// TwinCAT 3 PLC project ECRH
// ProgramVersion: 3.1.4023.0
// libraries:
//   Tc2_MBus, * (Beckhoff Automation GmbH)
//   Tc2_MC2, * (Beckhoff Automation GmbH)
//   Tc2_NC, * (Beckhoff Automation GmbH)
//   Tc2_Standard, * (Beckhoff Automation GmbH)
//   Tc2_System, * (Beckhoff Automation GmbH)
//   Tc3_Module, * (Beckhoff Automation GmbH)
// project tree:
//   GVLs/ GVL.TcGVL
//   / PlcTask.TcTTO
//   POUs/ MAIN.TcPOU, MAP.TcPOU, pCTRL_CODAC.TcPOU

CONFIGURATION ECRH
    RESOURCE PLC ON TwinCAT3
        TASK PlcTask(INTERVAL := T#10ms, PRIORITY := 20);
        PROGRAM MAIN WITH PlcTask : MAIN;
    END_RESOURCE
END_CONFIGURATION

// ---- GVLs/GVL.TcGVL
{attribute 'qualified_only'}
VAR_GLOBAL
	// Constantes de contrôle à ne pas dépasser
	dTemperature_Seuil_TBD : LREAL := 80000;
	dTension_Max : LREAL := 300;
	dCouple_Max : LREAL := 63 (*0.75 * 100 / 1.2*);
	
	// Peut-être à remplacer par les limites d'axes à définir dans MOTION -> Axes -> limit switches
	Butee_Min_M1X : LREAL := -49;
	Butee_Min_M1Y : LREAL := -17;
	Butee_Min_M2X : LREAL := -100;
	Butee_Min_M2Y : LREAL := -100;
	Butee_Min_M3X : LREAL := -100;
	Butee_Min_M3Y : LREAL := -100;
	Butee_Max_M1X : LREAL := 39;
	Butee_Max_M1Y : LREAL := 16;
	Butee_Max_M2X : LREAL := 100;
	Butee_Max_M2Y : LREAL := 100;
	Butee_Max_M3X : LREAL := 100;
	Butee_Max_M3Y : LREAL := 100;
	
	// Variable d'erreurs à envoyer au codac à intervalles de temps réguliers
	arrErrorSystem : ARRAY[0..4] OF BOOL := [FALSE, FALSE, FALSE, FALSE, FALSE];
	arrErrorTemperature : ARRAY[0..5] OF BOOL := [FALSE, FALSE, FALSE, FALSE, FALSE, FALSE];
	arrErrorTension : ARRAY[0..2] OF BOOL := [FALSE, FALSE, FALSE];
	arrErrorCouple : ARRAY[0..5] OF BOOL := [FALSE, FALSE, FALSE, FALSE];
	arrErrorPosition : ARRAY[0..5] OF BOOL := [FALSE, FALSE, FALSE, FALSE];
	
	// Variable qui stocke l'état de la commande moteur
	iEtatCmd : INT := 0;
	
	// Initialise la vitesse des moteurs
	dVelocite : LREAL := 10;
	dAcceleration : LREAL := 2;
	dDeceleration : LREAL := 2;
	dJerk : LREAL := 5000;
	
	// Définition des axes, doit être link aux axes du motion control
	M1_X : AXIS_REF;
	M1_Y : AXIS_REF;
	M2_X : AXIS_REF;
	M2_Y : AXIS_REF;
	M3_X : AXIS_REF;
	M3_Y : AXIS_REF;
	
	// Variable qui indique si une erreur est remarquée sur le système
	bError : BOOL := FALSE;
	
	// Variable qui définit la position voulue par le PCS
	dSetPosition_M1X : LREAL;
	dSetPosition_M1Y : LREAL;
	dSetPosition_M2X : LREAL;
	dSetPosition_M2Y : LREAL;
	dSetPosition_M3X : LREAL;
	dSetPosition_M3Y : LREAL;
	
	// Variable qui retient si une erreur est survenue lors de la dernière commande
	bErrorTwincat : BOOL;
	
	// Variable dont la valeur correspond à celle mesurée par le ThermoCouple indiqué
	arrTemperatures : ARRAY[0..5] OF LREAL;
	iTC1_M1 AT %I* : INT := 0;
	iTC2_M1 AT %I* : INT := 0;
	iTC1_M2 AT %I* : INT := 0;
	iTC2_M2 AT %I* : INT := 0;
	iTC1_M3 AT %I* : INT := 0;
	iTC2_M3 AT %I* : INT := 0;
		
	// Variable dont la valeur correspond à celle mesurée par le capteur de tension du câble
	arrTensions : ARRAY[0..2] OF LREAL;
	iTension_M1 AT %I* : INT := 0;
	iTension_M2 AT %I* : INT := 0;
	iTension_M3 AT %I* : INT := 0;
		
	// Variable à remplacer par la vrai variable qui indique si les moteurs sont arrêtés
	bMotor_Stopped : BOOL := FALSE;
	
	// Buffer qui contient les données d'intérêt des 200 dernières ms, ms étant l'index correspondant à la ms de l'instant t
	arrData : ARRAY [0..199] OF ARRAY[0..14] OF LREAL;
	ms : INT := 0;
	
	// Tableaux de données destinés à êtres récupérés par le CODAC -> faciliter l'accès aux données
	arrValues : ARRAY[0..14] OF LREAL;
	arrErrors : ARRAY[0..14] OF BOOL;
	arrButees : ARRAY[0..11] OF LREAL;
	
	// Détecteur placé proche de la butée mécanique pour permettre le homing de la position et avoir à partir de ce point un mouvement relatif connu
	bHomeSwitch_M1X AT %I*: BOOL;
	bHomeSwitch_M1Y AT %I*: BOOL;
	bHomeSwitch_M2X AT %I*: BOOL;
	bHomeSwitch_M2Y AT %I*: BOOL;
	bHomeSwitch_M3X AT %I*: BOOL;
	bHomeSwitch_M3Y AT %I*: BOOL;
	
	// Définit le mouvement à faire pour retomber sur une consigne moteur correspondant au 0° à partir de la position de homing
	dZero_M1X: LREAL;
	dZero_M1Y: LREAL;
	dZero_M2X: LREAL;
	dZero_M2Y: LREAL;
	dZero_M3X: LREAL;
	dZero_M3Y: LREAL;
	
	// Définit la commande de couple de chaque axe
	dSetTorque_M1X AT %Q*: UINT := 62;
	dSetTorque_M1Y AT %Q*: UINT := 62;
	dSetTorque_M2X AT %Q*: UINT := 62;
	dSetTorque_M2Y AT %Q*: UINT := 62;
	dSetTorque_M3X AT %Q*: UINT := 62;
	dSetTorque_M3Y AT %Q*: UINT := 62;
	
	// Boolean qui indique si l'initialisation est bien réalisée 
	bInit_OK: BOOL;

END_VAR

// ---- POUs/MAIN.TcPOU
PROGRAM MAIN
VAR
	Initialisation: INT := 0;
	En_Attente: INT := 100;
	En_Cours_De_Traitement: INT := 200;
	Stop: INT := 300;
	Reset: INT := 800;
	Erreur: INT := 900;
	
	McPower_M1X : MC_Power;
	McReset_M1X : MC_Reset;
	McStop_M1X : MC_Stop;
	McHome_M1X : MC_Home;
	McMoveAbs_M1X : MC_MoveAbsolute;
	
	McPower_M1Y : MC_Power;
	McReset_M1Y : MC_Reset;
	McStop_M1Y : MC_Stop;
	McHome_M1Y : MC_Home;
	McMoveAbs_M1Y : MC_MoveAbsolute;
END_VAR

// A chaque itération, il faut penser à appeler la fonction pour que son statut (Done, Busy, Error) se mette à jour
// Une façon de faire est d'appeler au début chaque fonction et de changer dans le corps du programme
// seulement le execute qui vaut true ou false
GVL.M1_X.ReadStatus();
McPower_M1X(Axis:=GVL.M1_X,Enable:=TRUE,Enable_Positive:=TRUE,Enable_Negative:=TRUE,Override:=100);
McReset_M1X(Axis:=GVL.M1_X);
McHome_M1X(Axis:=GVL.M1_X,bCalibrationCam := GVL.bHomeSwitch_M1X);
McMoveAbs_M1X(Axis:=GVL.M1_X);
McStop_M1X(Axis:=GVL.M1_X);

GVL.M1_Y.ReadStatus();
McPower_M1Y(Axis:=GVL.M1_Y,Enable:=TRUE,Enable_Positive:=TRUE,Enable_Negative:=TRUE,Override:=100);
McReset_M1Y(Axis:=GVL.M1_Y);
McHome_M1Y(Axis:=GVL.M1_Y,bCalibrationCam := GVL.bHomeSwitch_M1Y);
McMoveAbs_M1Y(Axis:=GVL.M1_Y);
McStop_M1Y(Axis:=GVL.M1_Y);

// Permet d'actualiser les données qui vont transités par ADS vers le CODAC
pCTRL_CODAC();

CASE GVL.iEtatCmd OF

	// INITIALISATION
	0: 
		// On commence par tout disable pour être sûr qu'il n'y ait pas d'erreur
		McReset_M1X(Axis:=GVL.M1_X, Execute:=FALSE);
		McHome_M1X(Axis:=GVL.M1_X,bCalibrationCam := GVL.bHomeSwitch_M1X, Execute:=FALSE);
		McMoveAbs_M1X(Axis:=GVL.M1_X, Execute:=FALSE);
		McStop_M1X(Axis:=GVL.M1_X, Execute:=FALSE);
		
		McReset_M1Y(Axis:=GVL.M1_Y, Execute:=FALSE);
		McHome_M1Y(Axis:=GVL.M1_Y,bCalibrationCam := GVL.bHomeSwitch_M1Y, Execute:=FALSE);
		McMoveAbs_M1Y(Axis:=GVL.M1_Y, Execute:=FALSE);
		McStop_M1Y(Axis:=GVL.M1_Y, Execute:=FALSE);
		
		// L'initialisation n'est pas faite donc on assigne FALSE
		GVL.bInit_OK := FALSE;
	
		// On commence par lancer un reset des axes
		McReset_M1X(Axis:= GVL.M1_X, Execute:= TRUE);
		McReset_M1Y(Axis:= GVL.M1_Y, Execute:= TRUE);
		IF GVL.bError OR McReset_M1X.Error OR McReset_M1Y.Error THEN
			GVL.iEtatCmd := Erreur;
		ELSE
			GVL.iEtatCmd := 5;				
		END_IF
		
		// On assigne au tableau de butées les valeurs à récupérer au CODAC
		GVL.arrButees[0]:=GVL.Butee_Min_M1X;
		GVL.arrButees[1]:=GVL.Butee_Max_M1X;
		GVL.arrButees[2]:=GVL.Butee_Min_M1Y;
		GVL.arrButees[3]:=GVL.Butee_Max_M1Y;
		GVL.arrButees[4]:=GVL.Butee_Min_M2X;
		GVL.arrButees[5]:=GVL.Butee_Max_M2X;
		GVL.arrButees[6]:=GVL.Butee_Min_M2Y;
		GVL.arrButees[7]:=GVL.Butee_Max_M2Y;
		GVL.arrButees[8]:=GVL.Butee_Min_M3X;
		GVL.arrButees[9]:=GVL.Butee_Max_M3X;
		GVL.arrButees[10]:=GVL.Butee_Min_M3Y;
		GVL.arrButees[11]:=GVL.Butee_Max_M3Y;
	
	// On attend la fin du reset
	5: 
		IF GVL.bError OR McReset_M1X.Error OR McReset_M1Y.Error THEN
			GVL.iEtatCmd := Erreur;
		ELSIF McReset_M1X.Done AND McReset_M1Y.Done THEN
			 GVL.iEtatCmd := 20;		
			McReset_M1X(Axis:= GVL.M1_X, Execute:= FALSE);
			McReset_M1Y(Axis:= GVL.M1_Y, Execute:= FALSE);		
		END_IF
		
	(* 10 réservée à la commande de limitation de couple originellement
	   finalement, celle-ci se réalise directement via la variable globale SetTorque
	   qui est linkée à bipolar torque limit au niveau du drive *)

	// On lance un homing général qui met le système au niveau du point connu avec la distance adaptée. 
	// La première fois, faire le homing jusqu'à 0 et déplacer le moteur jusqu'à la position de 0°
	// Configurer cette distance dans la calibration value sous M1_X -> Enc -> Homing -> Calibration value
	// Le 0 absolu est maintenant configuré au niveau du 0° et le homing arrive à -Dist
	20: 
		McHome_M1X(Axis:=GVL.M1_X, Execute:= TRUE, bCalibrationCam := GVL.bHomeSwitch_M1X, Position:= GVL.dZero_M1X);
		McHome_M1Y(Axis:=GVL.M1_Y, Execute:= TRUE, bCalibrationCam := GVL.bHomeSwitch_M1Y, Position:= GVL.dZero_M1Y);
		IF GVL.bError OR McHome_M1X.Error OR McHome_M1Y.Error THEN
			GVL.iEtatCmd := 900;
		ELSE
			GVL.iEtatCmd := 25;
		END_IF
			
	// On attend la fin du homing
	25: 
		IF McHome_M1Y.Error OR McHome_M1X.Error OR GVL.bError THEN
			GVL.iEtatCmd := Erreur;
		ELSIF McHome_M1X.Done AND McHome_M1Y.Done THEN
			McHome_M1X(Axis:= GVL.M1_X, Execute:= FALSE);
			McHome_M1Y(Axis:= GVL.M1_Y, Execute:= FALSE);
			GVL.iEtatCmd := 30;		
		END_IF
		
	// On fait un mouvement vers le 0 absolu  -- Seulement si la calibration value ne marche pas (30 à 50 inutile normalement)
	30: 
		McMoveAbs_M1X(Axis:=GVL.M1_X,
					Position:= 0,
					Velocity:= GVL.dVelocite,
					Acceleration:= GVL.dAcceleration,
					Deceleration:= GVL.dDeceleration,
					Jerk:= GVL.dJerk,
					Execute:= TRUE);
		McMoveAbs_M1Y(Axis:=GVL.M1_Y,
					Position:= 0,
					Velocity:= GVL.dVelocite,
					Acceleration:= GVL.dAcceleration,
					Deceleration:= GVL.dDeceleration,
					Jerk:= GVL.dJerk,
					Execute:= TRUE);
		IF GVL.bError OR McMoveAbs_M1X.Error OR McMoveAbs_M1Y.Error THEN
			GVL.iEtatCmd := 900;
		ELSE
			GVL.iEtatCmd := 35;
		END_IF
	
	35: // On attend le mouvement vers le 0 absolu
		IF McMoveAbs_M1Y.Error OR McMoveAbs_M1X.Error OR GVL.bError THEN
			GVL.iEtatCmd := Erreur;
		ELSIF McMoveAbs_M1X.Done AND McMoveAbs_M1Y.Done THEN
			McMoveAbs_M1X(Axis:= GVL.M1_X, Execute:= FALSE);
			McMoveAbs_M1Y(Axis:= GVL.M1_Y, Execute:= FALSE);
			GVL.bInit_OK:= TRUE;
			GVL.iEtatCmd := En_Attente;		
		END_IF
	
	100: // En attente d'un changement induit en ADS ou d'une erreur
		IF GVL.bError THEN
			GVL.iEtatCmd := Erreur;
		END_IF
		
	// Entâme de la phase de mouvement moteur : 
	// Déplacement moteur miroir en premier hors butees (PAS FORCEMENT NECESSAIRE) 
	// Déplacement cadre vers position voulue
	// Deplacement miroir vers position voulue
	// Retour en phase d'attente
	200:
		McMoveAbs_M1Y(Axis:=GVL.M1_Y,
					Position:= 0,
					Velocity:= GVL.dVelocite,
					Acceleration:= GVL.dAcceleration,
					Deceleration:= GVL.dDeceleration,
					Jerk:= GVL.dJerk,
					Execute:= TRUE);
		IF GVL.bError OR McMoveAbs_M1Y.Error THEN
			GVL.iEtatCmd := Erreur;
		ELSIF McMoveAbs_M1Y.Busy THEN
			GVL.iEtatCmd := 210;				
		END_IF
		
	210: // Attente du mouvement des miroirs à 0 mm
		IF McMoveAbs_M1Y.Error OR GVL.bError THEN
			GVL.iEtatCmd := Erreur;
		ELSIF McMoveAbs_M1Y.Done THEN
			McMoveAbs_M1Y(Axis:= GVL.M1_Y, Execute:= FALSE);
			GVL.iEtatCmd := 220;		
		END_IF
		
	220: // Déplacement du cadre à la position voulue
		McMoveAbs_M1X(Axis:=GVL.M1_X,
					Position:= GVL.dSetPosition_M1X,
					Velocity:= GVL.dVelocite,
					Acceleration:= GVL.dAcceleration,
					Deceleration:= GVL.dDeceleration,
					Jerk:= GVL.dJerk,
					Execute:= TRUE);
		IF GVL.bError OR McMoveAbs_M1X.Error THEN
			GVL.iEtatCmd := 900;
		ELSIF McMoveAbs_M1X.Busy THEN
			GVL.iEtatCmd := 230;
		END_IF
	
	230: // On attend la fin du mouvement
		IF McMoveAbs_M1X.Error OR GVL.bError THEN
			GVL.iEtatCmd := Erreur;
		ELSIF McMoveAbs_M1X.Done THEN
			McMoveAbs_M1X(Axis:= GVL.M1_X, Execute:= FALSE);
			GVL.iEtatCmd := 240;		
		END_IF
		
	240: // On déplace le miroir à la position voulue
		McMoveAbs_M1Y(Axis:=GVL.M1_Y,
					Position:= GVL.dSetPosition_M1Y,
					Velocity:= GVL.dVelocite,
					Acceleration:= GVL.dAcceleration,
					Deceleration:= GVL.dDeceleration,
					Jerk:= GVL.dJerk,
					Execute:= TRUE);
		IF GVL.bError OR McMoveAbs_M1Y.Error THEN
			GVL.iEtatCmd := Erreur;
		ELSE
			GVL.iEtatCmd := 250;				
		END_IF
		
	250: // On attend et on met en attente
		IF McMoveAbs_M1Y.Error OR GVL.bError THEN
			GVL.iEtatCmd := Erreur;
		ELSIF McMoveAbs_M1Y.Done THEN
			McMoveAbs_M1Y(Axis:= GVL.M1_Y, Execute:= FALSE);
			GVL.iEtatCmd := 100;		
		END_IF
	
	// Commande d'annulation de la commande moteurs
	// Pour cela on vient arrêter proprement le mouvement des moteurs via un stop
	300:
		McStop_M1X(Axis:=GVL.M1_X, Execute:=TRUE, Deceleration:=40, Jerk:=GVL.dJerk);
		McStop_M1Y(Axis:=GVL.M1_Y, Execute:=TRUE, Deceleration:=40, Jerk:=GVL.dJerk);
		IF GVL.bError OR McStop_M1Y.Error OR McStop_M1X.Error THEN
			GVL.iEtatCmd := Erreur;
		ELSIF McStop_M1Y.Busy AND McStop_M1X.Busy THEN
			GVL.iEtatCmd := 310;				
		END_IF
	
	// On attend la fin du stop et on oublie pas de disable le McMove pour ne pas que la commande reste active
	310:
		IF GVL.bError OR McStop_M1X.Error OR McStop_M1Y.Error THEN
			GVL.iEtatCmd := Erreur;
		ELSIF McStop_M1X.Done AND McStop_M1Y.Done THEN
			 GVL.iEtatCmd := 100;		
			McStop_M1X(Axis:= GVL.M1_X, Execute:= FALSE);
			McStop_M1Y(Axis:= GVL.M1_Y, Execute:= FALSE);	
			McMoveAbs_M1X(Axis:= GVL.M1_X, Execute := FALSE);
			McMoveAbs_M1Y(Axis:= GVL.M1_Y, Execute := FALSE);
		END_IF
		
	// On lance un reset général
	800:
		McReset_M1X(Axis:= GVL.M1_X, Execute:= TRUE);
		McReset_M1Y(Axis:= GVL.M1_Y, Execute:= TRUE);
		IF McReset_M1X.Error OR McReset_M1Y.Error THEN
			GVL.iEtatCmd := Erreur;
		ELSE
			GVL.iEtatCmd := 810;				
		END_IF
	
	// Lorsque celui-ci est effectué et si le système n'est pas en butée, on se met en attente
	810:
		IF McReset_M1X.Error OR McReset_M1Y.Error THEN
			GVL.iEtatCmd := Erreur;
		ELSIF McReset_M1X.Done AND McReset_M1Y.Done THEN		
			McReset_M1X(Axis:= GVL.M1_X, Execute:= FALSE);
			McReset_M1Y(Axis:= GVL.M1_Y, Execute:= FALSE);	
			IF GVL.arrErrorSystem[0] THEN
				GVL.iEtatCmd := 820;
			ELSE
				IF GVL.bInit_OK THEN
					GVL.iEtatCmd := 100;
				ELSE
					GVL.iEtatCmd := 20;
				END_IF
			END_IF
		END_IF
	
	// Si le système est en butée, on le sort des butées
	820:
		IF GVL.M1_X.NcToPlc.ActPos >= GVL.Butee_Max_M1X THEN
			McMoveAbs_M1X(Axis:=GVL.M1_X,
					Position:= GVL.Butee_Max_M1X - 5,
					Velocity:= GVL.dVelocite,
					Acceleration:= GVL.dAcceleration,
					Deceleration:= GVL.dDeceleration,
					Jerk:= GVL.dJerk,
					Execute:= TRUE);
		ELSIF GVL.M1_X.NcToPlc.ActPos <= GVL.Butee_Min_M1X THEN
			McMoveAbs_M1X(Axis:=GVL.M1_X,
					Position:= GVL.Butee_Min_M1X + 5,
					Velocity:= GVL.dVelocite,
					Acceleration:= GVL.dAcceleration,
					Deceleration:= GVL.dDeceleration,
					Jerk:= GVL.dJerk,
					Execute:= TRUE);
		ELSIF GVL.M1_Y.NcToPlc.ActPos <= GVL.Butee_Min_M1Y THEN
			McMoveAbs_M1Y(Axis:=GVL.M1_Y,
					Position:= GVL.Butee_Min_M1Y + 5,
					Velocity:= GVL.dVelocite,
					Acceleration:= GVL.dAcceleration,
					Deceleration:= GVL.dDeceleration,
					Jerk:= GVL.dJerk,
					Execute:= TRUE);
		ELSIF GVL.M1_Y.NcToPlc.ActPos >= GVL.Butee_Max_M1Y THEN
			McMoveAbs_M1Y(Axis:=GVL.M1_Y,
					Position:= GVL.Butee_Max_M1Y - 5,
					Velocity:= GVL.dVelocite,
					Acceleration:= GVL.dAcceleration,
					Deceleration:= GVL.dDeceleration,
					Jerk:= GVL.dJerk,
					Execute:= TRUE);
		END_IF
		GVL.iEtatCmd := 830;
	
	// On attend la sortie de la butée
	830:
		IF McMoveAbs_M1X.Error OR McMoveAbs_M1Y.Error THEN
			GVL.iEtatCmd := 900;
		ELSIF McMoveAbs_M1X.Done OR McMoveAbs_M1Y.Done THEN
			McMoveAbs_M1X(Axis:= GVL.M1_X, Execute:= FALSE);
			McMoveAbs_M1Y(Axis:= GVL.M1_Y, Execute:= FALSE);
			IF GVL.bInit_OK THEN
				GVL.iEtatCmd := 100;
			ELSE
				GVL.iEtatCmd := 20;
			END_IF
		END_IF
		
	// Traitement de l'erreur
	900:
		IF GVL.arrErrorSystem[0] THEN
			GVL.iEtatCmd := 910;
		ELSE
			GVL.iEtatCmd := 990;
		END_IF
		
	// Erreur liée à la position, on arrête vite les moteurs pour ne pas forcer sur la butée
	910:
		McStop_M1X(Axis:=GVL.M1_X, Execute:=TRUE, Deceleration:=40, Jerk:=GVL.dJerk);
		McStop_M1Y(Axis:=GVL.M1_Y, Execute:=TRUE, Deceleration:=40, Jerk:=GVL.dJerk);
		IF McStop_M1X.Error OR McStop_M1X.Error THEN
			GVL.iEtatCmd := 990;
		ELSIF McStop_M1X.Busy AND McStop_M1Y.Busy THEN
			GVL.iEtatCmd := 920;
		END_IF
	
	// Lorsque c'est fait on se place dans l'état d'erreur général
	920:
		IF McStop_M1X.Error OR McStop_M1Y.Error THEN
			GVL.iEtatCmd := Erreur;
		ELSIF McStop_M1X.Done AND McStop_M1Y.Done THEN
			GVL.iEtatCmd := 990;		
			McStop_M1X(Axis:= GVL.M1_X, Execute:= FALSE);
			McStop_M1Y(Axis:= GVL.M1_Y, Execute:= FALSE);	
			McMoveAbs_M1X(Axis:= GVL.M1_X, Execute := FALSE);
			McMoveAbs_M1Y(Axis:= GVL.M1_Y, Execute := FALSE);
		END_IF
	
	// Etat général d'erreur dans lequel on disable tout et on attend une action par le CODAC 
	990:
		McReset_M1X(Axis:=GVL.M1_X, Execute:=FALSE);
		McHome_M1X(Axis:=GVL.M1_X,bCalibrationCam := GVL.bHomeSwitch_M1X, Execute:=FALSE);
		McMoveAbs_M1X(Axis:=GVL.M1_X, Execute:=FALSE);
		McStop_M1X(Axis:=GVL.M1_X, Execute:=FALSE);
		
		McReset_M1Y(Axis:=GVL.M1_Y, Execute:=FALSE);
		McHome_M1Y(Axis:=GVL.M1_Y,bCalibrationCam := GVL.bHomeSwitch_M1Y, Execute:=FALSE);
		McMoveAbs_M1Y(Axis:=GVL.M1_Y, Execute:=FALSE);
		McStop_M1Y(Axis:=GVL.M1_Y, Execute:=FALSE);
		
END_CASE

END_PROGRAM

// ---- POUs/pCTRL_CODAC.TcPOU
// Procédure qui met à jour toutes les variables que le CODAC vient récupérer
// Pour l'instant, le CODAC récupère seulement les valeurs de l'instant t mais il faudra peut-être penser à faire un buffer pour stocker les valeurs non récupérées
PROGRAM pCTRL_CODAC
VAR
END_VAR

// Actualise les deux variables à récupérer
METH_arrValues_actualisation();
METH_arrErrors_actualisation();
METH_arrData_actualisation();

METHOD METH_arrData_actualisation : BOOL
VAR_INPUT
END_VAR

VAR
	i: INT;
END_VAR
FOR i := 0 TO 15 DO
	GVL.arrData[GVL.ms][i] := GVL.arrValues[i];
END_FOR

IF GVL.ms < 199 THEN
	GVL.ms := GVL.ms + 1;
ELSE
	GVL.ms := 0;
END_IF
END_METHOD

// Méthode qui actualise le tableau arrErrors
METHOD METH_arrErrors_actualisation : BOOL
VAR_INPUT
END_VAR
VAR
	i : INT;
END_VAR
// Enregistre dans chaque case du tableau la donnée d'un capteur de température
// à savoir si la valeur mesurée est supérieure (true) ou inférieure (false) au seuil TBD
FOR i := 0 TO 5 DO
	GVL.arrErrorTemperature[i] := GVL.arrTemperatures[i] > GVL.dTemperature_Seuil_TBD;
END_FOR

// Enregistre dans chaque case du tableau la donnée d'un capteur de tension
FOR i := 0 TO 2 DO
	GVL.arrErrorTension[i] := GVL.arrTensions[i] > GVL.dTension_Max;
END_FOR

// Enregistre dans chaque case du tableau la donnée du couple mesurée par le moteur
GVL.arrErrorCouple[0] := GVL.M1_X.NcToPlc.ActTorque > GVL.dCouple_Max;
GVL.arrErrorCouple[1] := GVL.M1_Y.NcToPlc.ActTorque > GVL.dCouple_Max;
GVL.arrErrorCouple[2] := GVL.M2_X.NcToPlc.ActTorque > GVL.dCouple_Max;
GVL.arrErrorCouple[3] := GVL.M2_Y.NcToPlc.ActTorque > GVL.dCouple_Max;
GVL.arrErrorCouple[4] := GVL.M3_X.NcToPlc.ActTorque > GVL.dCouple_Max;
GVL.arrErrorCouple[5] := GVL.M3_Y.NcToPlc.ActTorque > GVL.dCouple_Max;


// Enregistre dans chaque case du tableau la donnée de la position par rapport aux butées
IF GVL.bInit_OK THEN
	GVL.arrErrorPosition[0] := GVL.M1_X.NcToPlc.ActPos < GVL.Butee_Min_M1X OR GVL.M1_X.NcToPlc.ActPos > GVL.Butee_Max_M1X;
	GVL.arrErrorPosition[1] := GVL.M1_Y.NcToPlc.ActPos < GVL.Butee_Min_M1Y OR GVL.M1_Y.NcToPlc.ActPos > GVL.Butee_Max_M1Y;
	GVL.arrErrorPosition[2] := GVL.M2_X.NcToPlc.ActPos < GVL.Butee_Min_M2X OR GVL.M2_X.NcToPlc.ActPos > GVL.Butee_Max_M2X;
	GVL.arrErrorPosition[3] := GVL.M2_Y.NcToPlc.ActPos < GVL.Butee_Min_M2Y OR GVL.M2_Y.NcToPlc.ActPos > GVL.Butee_Max_M2Y;
	GVL.arrErrorPosition[4] := GVL.M2_X.NcToPlc.ActPos < GVL.Butee_Min_M2X OR GVL.M2_X.NcToPlc.ActPos > GVL.Butee_Max_M2X;
	GVL.arrErrorPosition[5] := GVL.M2_Y.NcToPlc.ActPos < GVL.Butee_Min_M2Y OR GVL.M2_Y.NcToPlc.ActPos > GVL.Butee_Max_M2Y;
ELSE
	GVL.arrErrorPosition[0] := FALSE;
	GVL.arrErrorPosition[1] := FALSE;
	GVL.arrErrorPosition[2] := FALSE;
	GVL.arrErrorPosition[3] := FALSE;
	GVL.arrErrorPosition[4] := FALSE;
	GVL.arrErrorPosition[5] := FALSE;
END_IF

// Enregistre dans chaque case du tableau la donnée d'un groupe de contrôle - position, couple, tension ou température
GVL.arrErrorSystem[0] := GVL.arrErrorPosition[0] OR GVL.arrErrorPosition[1] OR GVL.arrErrorPosition[2] OR GVL.arrErrorPosition[3] OR GVL.arrErrorPosition[4] OR GVL.arrErrorPosition[5] ;
GVL.arrErrorSystem[1] := GVL.arrErrorCouple[0] OR GVL.arrErrorCouple[1] OR GVL.arrErrorCouple[2] OR GVL.arrErrorCouple[3] OR GVL.arrErrorCouple[4] OR GVL.arrErrorCouple[5]; 
GVL.arrErrorSystem[2] := GVL.arrErrorTension[0] OR GVL.arrErrorTension[1] OR GVL.arrErrorTension[2];
GVL.arrErrorSystem[3] := GVL.arrErrorTemperature[0] OR GVL.arrErrorTemperature[1] OR GVL.arrErrorTemperature[2] OR GVL.arrErrorTemperature[3] 
OR GVL.arrErrorTemperature[4] OR GVL.arrErrorTemperature[5];
GVL.arrErrorSystem[4] := GVL.M1_X.Status.Error OR GVL.M1_Y.Status.Error OR GVL.M2_X.Status.Error OR GVL.M2_Y.Status.Error
OR GVL.M3_X.Status.Error OR GVL.M3_Y.Status.Error;
 
// Enregistre sur une seule variable s'il y a une erreur ou pas
GVL.bError := GVL.arrErrorSystem[0] OR GVL.arrErrorSystem[1] OR GVL.arrErrorSystem[2] OR GVL.arrErrorSystem[3] OR GVL.arrErrorSystem[4];

// Compile l'ensemble des variables en un seul tableau pour transiter les données plus facilement
FOR i := 0 TO 5 DO
	GVL.arrErrors[i] := GVL.arrErrorTemperature[i];
END_FOR

FOR i := 0 TO 2 DO
	GVL.arrErrors[6+i] := GVL.arrErrorTension[i];
END_FOR

FOR i := 0 TO 5 DO
	GVL.arrErrors[9+i] := GVL.arrErrorPosition[i];
END_FOR
END_METHOD

// Méthode qui actualise le tableau arrValues
METHOD METH_arrValues_actualisation : BOOL
VAR_INPUT
END_VAR
VAR
	i : INT;
END_VAR
GVL.arrTemperatures[0] := MAP(GVL.iTC1_M1, 0, 65535, 0, 65535*0.1);
GVL.arrTemperatures[1] := MAP(GVL.iTC2_M1, 0, 65535, 0, 65535*0.1);
GVL.arrTemperatures[2] := MAP(GVL.iTC1_M2, 0, 65535, 0, 65535*0.1);
GVL.arrTemperatures[3] := MAP(GVL.iTC2_M2, 0, 65535, 0, 65535*0.1);
GVL.arrTemperatures[4] := MAP(GVL.iTC1_M3, 0, 65535, 0, 65535*0.1);
GVL.arrTemperatures[5] := MAP(GVL.iTC2_M3, 0, 65535, 0, 65535*0.1);

GVL.arrTensions[0] := MAP(GVL.iTension_M1, -32767, 32767, -10, 10);
GVL.arrTensions[1] := MAP(GVL.iTension_M2, -32767, 32767, -10, 10);
GVL.arrTensions[2] := MAP(GVL.iTension_M3, -32767, 32767, -10, 10); 

// associe à chaque case du tableau une valeur d'intérêt pour le CODAC
FOR i := 0 TO 5 DO
	GVL.arrValues[i] := GVL.arrTemperatures[i];
END_FOR

FOR i := 0 TO 2 DO
	GVL.arrValues[6+i] := GVL.arrTensions[i];
END_FOR

GVL.arrValues[9]  := GVL.M1_X.NcToPlc.ActPos;
GVL.arrValues[10] := GVL.M1_Y.NcToPlc.ActPos;
GVL.arrValues[11] := GVL.M2_X.NcToPlc.ActPos;
GVL.arrValues[12] := GVL.M2_Y.NcToPlc.ActPos;
GVL.arrValues[13] := GVL.M3_X.NcToPlc.ActPos;
GVL.arrValues[14] := GVL.M3_Y.NcToPlc.ActPos;
END_METHOD

END_PROGRAM

// ---- POUs/MAP.TcPOU
// Remet à a bonne échelle, map identique à celui d'arduino
FUNCTION MAP : LREAL
VAR_INPUT
	x : LREAL;
	in_min : LREAL;
	in_max : LREAL;
	out_min : LREAL;
	out_max : LREAL;
	
END_VAR
VAR
END_VAR


IF ((in_max - in_min) + out_min) <> 0 THEN
	MAP := (x - in_min) * (out_max - out_min) / (in_max - in_min) + out_min;
ELSE
	MAP := 0;
END_IF

RETURN;

END_FUNCTION
